{attribute 'qualified_only'}
VAR_GLOBAL
	aOutputSolValve 		: ARRAY[1..GVL_CONSTANT.NumSolValve] OF BOOL; //Solenoid Valve
	aAnalogController 		: ARRAY[1..GVL_CONSTANT.NumAnalogController] OF AnalogController; //Flow Controller (Ramp Controller) for MFC, EPC, Reactor
	aMaxValue		: ARRAY[1..GVL_CONSTANT.NumAnalogController] OF REAL; //Max Value set from UI Application
	
	(* Present Value Meter Display*)
	aMonitoring_PV 			: ARRAY[1..GVL_CONSTANT.NumMonitoring] OF REAL; //Gauge Monitoring Value to UI
	
	interlock 				: Interlock;
	generalIO				: GeneralIO;
	mainPRGControl : MainPRGControl;
	recipe :Recipe;
END_VAR

(* stored: Version 1.1.0.1, ProductVersion 3.1.4026.11
   GVL GVL_INTERFACE_UI: Id {39e04069-2aa1-47f6-95f8-4e7243c4d4fa} *)
